{attribute 'linkalways'} 
{attribute 'no_explicit_call' := 'This FB is a CLASS and must be accessed using methods or properties'}
{attribute 'enable_dynamic_creation'}
FUNCTION_BLOCK FINAL XOR_WORD EXTENDS Node
VAR
	in1 : _WORD(0);
	in2 : _WORD(0);
	out : _WORD(0);
END_VAR

METHOD PUBLIC Clone : I_Node
VAR
	pNode : POINTER TO XOR_WORD;
END_VAR
pNode := __NEW(XOR_WORD);
Clone := pNode^;
END_METHOD

METHOD FB_init : BOOL
VAR_INPUT
	bInitRetains : BOOL; // if TRUE, the retain variables are initialized (warm start / cold start)
	bInCopyCode : BOOL;  // if TRUE, the instance afterwards gets moved into the copy code (online change)
END_VAR
AddInput('in1',THIS^.in1);
AddInput('in2',THIS^.in2);
AddOutput('out', THIS^.out);
END_METHOD

METHOD PROTECTED OnExecute
VAR
END_VAR
out.Value := in1.Value XOR in2.Value;
END_METHOD

END_FUNCTION_BLOCK

(* stored: Version 1.1.0.1, ProductVersion 3.1.4024.15
   POU XOR_WORD: Id {733ec959-17b4-4529-a474-deabd9f90d9c}, SpecialFunc None
   Folder Constructor: Id {e3267c38-5da3-4255-a6c1-bf91a902fe51}
   Method Clone: Id {410edd79-8ad7-46e5-b2ec-c528c2f8d7f8}
   Method FB_init: Id {7ec1a9d9-85c7-41b3-b2c5-7edcc041486a}
   Method OnExecute: Id {21941262-460f-4e0b-a722-3628adb14cf3} *)
